(* PLC project Recipe_Tool, Beckhoff Automation GmbH TwinCAT PLC Control 3.5.3.40 *)
(* stored: creationDateTime 2014-11-23T03:47:42.5228328, modificationDateTime 2014-11-23T03:47:42.5228328 *)

TYPE DUT_RecipeCommand : STRUCT
  SkillID : INT;
  SkillName : STRING(80);
  Quantity : LREAL;
END_STRUCT;
END_TYPE
